// TwinCAT 3 PLC project segmentationDL
// ProgramVersion: 3.1.4026.10
// libraries:
//   Tc2_Standard, * (Beckhoff Automation GmbH)
//   Tc2_System, * (Beckhoff Automation GmbH)
//   Tc3_MlServer, * (Beckhoff Automation GmbH)
//   Tc3_Vision, * (Beckhoff Automation GmbH)
// project tree:
//   DUTs/ ST_modelInput.TcDUT, ST_modelOutput.TcDUT
//   GVLs/ constants.TcGVL
//   / PlcTask.TcTTO
//   POUs/Functions/ binarizeSegmentationMatrixFunction.TcPOU, contourSegmentationFunction.TcPOU, convertToBwFunction.TcPOU, flattenSegmentationMatrixFunction.TcPOU, imageNormalizationFunction.TcPOU, imageTilingFunction.TcPOU, imageToMatrixFunction.TcPOU, matrixToMaskFunction.TcPOU, nnPredictFunction.TcPOU, readImageFunction.TcPOU, reassembleImageFunction.TcPOU
//   POUs/Functions/Other/ binarizeSegmentationImageFunction.TcPOU, extractSingleTileFunction.TcPOU, flattenedTileToImageFunction.TcPOU, flattenMatrixFunction.TcPOU, flattenTileFunction.TcPOU, matrixToImageFunction.TcPOU
//   POUs/ MAIN.TcPOU
// real-time tasks:
//   TASK PlcTask: cycle T#10ms, priority 20, ADS port 350

CONFIGURATION segmentationDL
    RESOURCE PLC ON TwinCAT3
        TASK PlcTask(INTERVAL := T#10ms, PRIORITY := 20);
        PROGRAM MAIN WITH PlcTask : MAIN;
    END_RESOURCE
END_CONFIGURATION

// ---- DUTs/ST_modelInput.TcDUT
TYPE ST_modelInput :
STRUCT

	{attribute 'hide'} _header_DO_NOT_CHANGE : ARRAY[0..63] OF SINT := [-1,-112,120,86,52,18,-1,-1,1,-1,0,0,-1,-1,-112,-112,5,-37,-120,51,81,-94,-125,-64,-81,-119,-103,-51,-65,-118,48,-32,-5,44,-121,-88,-37,0,73,-109,92,-4,-120,92,99,42,-107,-53,64,-52,3,0,0,0,0,0,0,0,0,0,0,0,0,0];
	in_args_0 : ARRAY[0..0,0..287,0..215,0..0] OF REAL;

END_STRUCT
END_TYPE

// ---- DUTs/ST_modelOutput.TcDUT
TYPE ST_modelOutput :
STRUCT

	{attribute 'hide'} _header_DO_NOT_CHANGE : ARRAY[0..63] OF SINT := [-1,-112,120,86,52,18,-1,-1,1,-1,0,0,-1,-1,-112,-112,5,-37,-120,51,81,-94,-125,-64,-81,-119,-103,-51,-65,-118,48,-32,-5,44,-121,-88,-37,0,73,-109,92,-4,-120,92,99,42,-107,-53,64,-52,3,0,0,0,0,0,0,0,0,0,0,0,0,0];
	out_conv2d_14 : ARRAY[0..0,0..287,0..215,0..0] OF REAL;

END_STRUCT
END_TYPE

// ---- GVLs/constants.TcGVL
{attribute 'qualified_only'}
VAR_GLOBAL CONSTANT
	
	// Dimensions of the image
	IMG_WIDTH: UDINT := 1080;
	IMG_HEIGHT: UDINT := 1440;
	
	// Dimensions of the tile
	TILE_WIDTH: UDINT := 216;
	TILE_HEIGHT: UDINT := 288;
	
	// Total number of tiles
	NUM_TILES: UDINT := 25; 
	
END_VAR

// ---- POUs/MAIN.TcPOU
PROGRAM MAIN
VAR
	
	filePath: STRING := 'C:\Users\UserName\Desktop\visionFiles\images\000188.jpg'; // Change accordingly
	
	modelFilePath: STRING := 'C:\Users\UserName\Desktop\visionFiles\model\model.json'; // Change accordingly
	
	// Processing chain
	readImage: readImageFunction;
	convertToBw: convertToBwFunction;
	imageToMatrix: imageToMatrixFunction;
	imageNormalization: imageNormalizationFunction;
	imageTiling: imageTilingFunction;
	nnPredict: nnPredictFunction;
	reassembleImage: reassembleImageFunction;
	matrixToMask: matrixToMaskFunction;
	binarizeSegmentationMatrix: binarizeSegmentationMatrixFunction;
	contourSegmentation: contourSegmentationFunction;
	
	image: ITcVnImage;
	imageDisp: ITcVnDisplayableImage;
	
	segmentation: ITcVnImage;
	segmentationDisp: ITcVnDisplayableImage;
	
	contours: ITcVnImage;
	contoursDisp: ITcVnDisplayableImage;

	
	imageMatrix: ARRAY[1..constants.IMG_WIDTH, 1..constants.IMG_HEIGHT] OF REAL;
	tiles: ARRAY[1..constants.NUM_TILES, 1..constants.TILE_WIDTH, 1..constants.TILE_HEIGHT] OF REAL;
	
	segmentationTiles: ARRAY[1..constants.NUM_TILES, 1..constants.TILE_WIDTH, 1..constants.TILE_HEIGHT] OF REAL;
	segmentationMatrix: ARRAY[1..constants.IMG_WIDTH, 1..constants.IMG_HEIGHT] OF REAL;
	segmentationMatixBinarized: ARRAY[1..constants.IMG_WIDTH, 1..constants.IMG_HEIGHT] OF USINT;
	
	error: BOOL;
	hResult: HRESULT;

END_VAR

// Read the image
readImage(filePath := filePath,
		  image := image,
		  imageDisp := imageDisp,
		  error => error);
		  
// Convert the image to Black and White
convertToBw(image := image,
			imageDisp := imageDisp,
			start := readImage.finished,
			error => error);

// Extract the image values in the form of a matrix
imageToMatrix(image := image,
			  start := convertToBw.finished,
			  imageMatrix := imageMatrix,
			  error => error);

// Normalize image values from 0->255 to 0->1		  
imageNormalization(imageMatrix := imageMatrix,
					start := imageToMatrix.finished,
					error => error);
					
// Tile the image			  
imageTiling(tiles := tiles,
			imageMatrix := imageMatrix,
			start := imageNormalization.finished);
					
// Neural Network prediction
nnPredict(tiles := tiles,
		  modelFilePath := modelFilePath,
		  start := imageTiling.finished,
		  segmentationTiles => segmentationTiles);

// Reassembling tiles into an image matrix
reassembleImage(tiles := segmentationTiles,
				start := nnPredict.finished,
				imageMatrix => segmentationMatrix);
				
// Binarize the output of the neural network
binarizeSegmentationMatrix(segmentationMatrix := segmentationMatrix,
						   segmentationMatrixBinarized := segmentationMatixBinarized,
						   start := reassembleImage.finished);

// Use this to convert the segmentation matrix into a usable twincat image
matrixToMask(matrix := segmentationMatixBinarized,
			 image := segmentation,
			 imageDisp := segmentationDisp,
			 start := 	binarizeSegmentationMatrix.finished,
			 error => error);

// Plot the contour overlaid 
contourSegmentation(image := image,
					segmentationImage := segmentation,
					contoursImage := contours,
					contoursImageDisp := contoursDisp,
					minimumArea := 100,
					start := matrixToMask.finished,);

END_PROGRAM

// ---- POUs/Functions/readImageFunction.TcPOU
FUNCTION_BLOCK readImageFunction

VAR_IN_OUT
	image: ITcVnImage;
	imageDisp: ITcVnDisplayableImage;
END_VAR

VAR_INPUT
	filePath: STRING;
END_VAR

VAR_OUTPUT
	error: BOOL;
	finished: BOOL;
END_VAR


VAR
	readImageTrg: F_TRIG;	

	readImage: FB_VN_ReadImage;
	readImageCmd: BOOL := TRUE;
	
	imageRef: REFERENCE TO ITcVnImage;
	imageDispRef: REFERENCE TO ITcVnDisplayableImage;
	
	hResult: HRESULT;
	isImageRead: BOOL;
END_VAR

// Assign references
imageRef REF= image;
imageDispRef REF= imageDisp;

// Read the image
readImage(sFilePath := filePath,
          ipDestimage := imageRef,
          bRead := readImageCmd);
		 
// Trigger on when the image is read
readImageTrg(CLK := readImage.bBusy);

// If there is an error, latch onto it
IF readImage.bError THEN
    error := TRUE;
END_IF

// Reset the command after execution if needed for edge triggering
IF readImage.bBusy THEN
    readImageCmd := FALSE;
END_IF

// Raise a flag when the image has been read
IF (readImageTrg.Q) AND (NOT error) THEN
	isImageRead := TRUE;
END_IF

// Convert to a displayable image to view in the ADS Image View, if possible
IF (NOT error) AND (isImageRead) AND (NOT finished) THEN
	
    // Copy the image into a displayable one so that we can access it via the ADS Image Watch
    hResult := F_VN_CopyIntoDisplayableImage(ipSrcImage := image,
                                             ipDestImage := imageDispRef,
                                             hrPrev := hResult);

	// If there is an error, latch onto it
    IF FAILED(hResult) THEN
        error := TRUE;
    END_IF
	
	IF SUCCEEDED(hResult) THEN
		finished := TRUE;
	END_IF
	
END_IF

END_FUNCTION_BLOCK

// ---- POUs/Functions/convertToBwFunction.TcPOU
FUNCTION_BLOCK convertToBwFunction

VAR_IN_OUT
	image: ITcVnImage;
	imageDisp: ITcVnDisplayableImage;
END_VAR

VAR_INPUT
	start: BOOL;
END_VAR

VAR_OUTPUT
	error: BOOL;
	finished: BOOL := FALSE;
END_VAR


VAR

	originalImage: ITcVnImage;

	imageRef: REFERENCE TO ITcVnImage;
	imageDispRef: REFERENCE TO ITcVnDisplayableImage;
	
	hResult: HRESULT;
END_VAR

// Assign references
imageRef REF= image;
imageDispRef REF= imageDisp;
	
IF (start) AND (NOT error) AND (NOT finished) THEN
	
	originalImage := image;

	// Convert to black and white
	hResult := F_VN_ConvertColorSpace(ipSrcImage := image,
										ipDestImage := imageRef,
										eTransform := ETcVnColorSpaceTransform.TCVN_CST_RGB_TO_GRAY,
										hrPrev := hResult);
										
	// If there is an error, latch onto it
    IF FAILED(hResult) THEN
        error := TRUE;
    END_IF
	
	IF SUCCEEDED(hResult) THEN
		
		 // Copy the image into a displayable one so that we can access it via the ADS Image Watch
		hResult := F_VN_CopyIntoDisplayableImage(ipSrcImage := image,
											    	ipDestImage := imageDispRef,
											    	hrPrev := hResult);
	
		// If there is an error, latch onto it
		IF FAILED(hResult) THEN
			error := TRUE;
		END_IF
		
		IF SUCCEEDED(hResult) THEN
			finished := TRUE;
		END_IF
		
	END_IF
	
END_IF

END_FUNCTION_BLOCK

// ---- POUs/Functions/imageToMatrixFunction.TcPOU
FUNCTION_BLOCK imageToMatrixFunction

// See: https://infosys.beckhoff.com/english.php?content=../content/1033/tf7xxx_tc3_vision/6997345803.html&id=

VAR_IN_OUT
	imageMatrix: ARRAY[1..constants.IMG_WIDTH, 1..constants.IMG_HEIGHT] OF REAL;
END_VAR

VAR_INPUT
	image: ITcVnImage;
	start: BOOL;
END_VAR

VAR_OUTPUT
	error: BOOL;
	finished: BOOL := FALSE;
END_VAR

VAR
	
    nHeight     :   UDINT;
    nWidth      :   UDINT;
    y           :   UDINT;
    x           :   UDINT;
	
    pRow        :   POINTER TO USINT;
    nPixelValue :   USINT;
	
	hResult: HRESULT;
	
END_VAR

	
IF start AND (NOT finished) THEN
	
	// Retrieve the image width and height
	//hResult := F_VN_GetImageWidth(image, nWidth, hResult);
	//hResult := F_VN_GetImageHeight(image, nHeight, hResult);
	
	// Iterate every pixel of the image
	
	
	FOR y := 0 TO constants.IMG_HEIGHT - 1 DO
	
		// Get the pointer to the image row
		HRESULT := image.GetRowPointer(y, ADR(pRow));
		
		FOR x := 0 TO constants.IMG_WIDTH - 1 DO
			
			// Access the single pixel value
			nPixelValue := pRow[x]; 
			
			// Assign the pixel value to the image matrix
			imageMatrix[x+1, y+1] := nPixelValue; 
			
		END_FOR
	
		// It’s important to release the pointer. Otherwise there will be memory leaks.
		HRESULT := image.ReleaseRowPointer(ADR(pRow)); 
		
	END_FOR

	finished := TRUE;

END_IF

END_FUNCTION_BLOCK

// ---- POUs/Functions/imageNormalizationFunction.TcPOU
FUNCTION_BLOCK imageNormalizationFunction

VAR_IN_OUT
	imageMatrix: ARRAY[1..constants.IMG_WIDTH, 1..constants.IMG_HEIGHT] OF REAL;
END_VAR

VAR_INPUT
	start: BOOL;
END_VAR

VAR_OUTPUT
	error: BOOL;
	finished: BOOL := FALSE;
END_VAR

VAR
	x: UDINT;
	y: UDINT;
	normalizationFactor: REAL := 255.0;
END_VAR

	
IF (start) AND (NOT finished) THEN
	
	FOR x := 1 TO constants.IMG_WIDTH DO
		FOR y := 1 TO constants.IMG_HEIGHT DO
			
			imageMatrix[x, y] := imageMatrix[x, y] / normalizationfactor;
			
		END_FOR
	END_FOR
	
	finished := TRUE;
	 
END_IF

END_FUNCTION_BLOCK

// ---- POUs/Functions/imageTilingFunction.TcPOU
FUNCTION_BLOCK imageTilingFunction

VAR_IN_OUT
	tiles: ARRAY[1..constants.NUM_TILES, 1..constants.TILE_WIDTH, 1..constants.TILE_HEIGHT] OF REAL;
	start: BOOL;
END_VAR

VAR_INPUT
    imageMatrix: ARRAY[1..constants.IMG_WIDTH, 1..constants.IMG_HEIGHT] OF REAL;
END_VAR

VAR_OUTPUT
	finished: BOOL;
END_VAR

VAR
    tileRow: UDINT; // Row of the tile grid
    tileCol: UDINT; // Column of the tile grid
    currentTile: UDINT; // Counter for the tiles
    
    startX: UDINT; // X coordinate for the start of the tile
    startY: UDINT; // Y coordinate for the start of the tile
    X: UDINT; // X position within the tile
    Y: UDINT; // Y position within the tile
	
	nTilesHorizontal: UDINT;
	nTilesVertical: UDINT;
	
	
    
END_VAR


IF start AND NOT finished THEN
	
	// We start from the first tile
	currentTile := 1;
	
	// Finding how many tiles in the horizontal and vertical direction
	nTilesVertical := constants.IMG_HEIGHT / constants.TILE_HEIGHT;
	nTilesHorizontal := constants.IMG_WIDTH / constants.TILE_WIDTH;
	
	
	// Cycling on the tiles
	
	// Y
	FOR tileRow := 1 TO nTilesVertical DO
		
		// X
		FOR tileCol := 1 TO nTilesHorizontal DO
	
			// Determining the top left point coordinate of each tile
			startY := (tileRow - 1) * constants.TILE_HEIGHT + 1;
			startX := (tileCol - 1) * constants.TILE_WIDTH + 1;
			
			// Cycling on the pixels of the tile
			FOR X := 1 TO constants.TILE_WIDTH DO
				FOR Y := 1 TO constants.TILE_HEIGHT DO
					tiles[currentTile, X, Y] := imageMatrix[startX + X - 1, startY + Y - 1]; // Subtract 1 since the inner for loops add 1
				END_FOR
			END_FOR
	
			// Update the current tile
			currentTile := currentTile + 1;
	
		END_FOR
	END_FOR

	finished := TRUE;

END_IF

END_FUNCTION_BLOCK

// ---- POUs/Functions/nnPredictFunction.TcPOU
FUNCTION_BLOCK nnPredictFunction

// see: https://infosys.beckhoff.com/english.php?content=../content/1033/tf3820_tc3_machine_learning_server/17276127115.html&id=9003034378846799115

VAR_INPUT
	tiles: ARRAY[1..constants.NUM_TILES, 1..constants.TILE_WIDTH, 1..constants.TILE_HEIGHT] OF REAL;
	modelFilePath: STRING;
	start: BOOL;
END_VAR

VAR_OUTPUT
	segmentationTiles: ARRAY[1..constants.NUM_TILES, 1..constants.TILE_WIDTH, 1..constants.TILE_HEIGHT] OF REAL;
	finished: BOOL;
	error: BOOL;
END_VAR

VAR

	stModelInput: ST_modelInput;
	stModelOutput: ST_modelOutput;

	fbMlSvr: FB_MlSvrPrediction;
	
	n: UDINT := 1;
	x: UDINT;
	y: UDINT;
	
	nextTile: BOOL := TRUE;
	
END_VAR

// ===================================
// 1. Configuring the ML server
// ===================================

// Path to model  
fbMlSvr.stPredictionParameter.sMlModelFilePath := modelFilePath;

 // We want to execute the model on localsystem --> localhost                                     
fbMlSvr.stPredictionParameter.sMlSvrNetId := '127.0.0.1.1.1';

// Where to execute the model --> CPU
fbMlSVr.stPredictionParameter.eExecutionProvider := E_EXECUTIONPROVIDER.CPU; 

// Submit configuration request to the TcMlServer
fbMlSvr.Configure(nTimeout := 1000, nPriority:=0);

IF (fbMlSvr.bError) THEN
	error := TRUE;
END_IF


// ===================================================
// 2. Use the model for predictions
// ===================================================

// If the server is configured
IF (fbMlSvr.bConfigured) AND (start) AND (NOT finished) THEN
	
	// Cycling on the tiles, use an IF statement since it can take multiple PLC cycles
	IF n <= constants.NUM_TILES THEN
		
		// If it is time to process the next tile
		IF nextTile THEN
			
			nextTile := FALSE;
			
			// Format the tile for the model input
			FOR y := 1 TO constants.TILE_HEIGHT DO
				FOR x := 1 TO constants.TILE_WIDTH DO
					stModelInput.in_args_0[0, y-1, x-1, 0] := tiles[n, x, y];
				END_FOR
			END_FOR
			
		END_IF
		
		// Predict
		IF fbMlSvr.Predict(pDataIn := ADR(stModelInput), 
						   nDataInSize := SIZEOF(stModelInput), 
						   pDataOut := ADR(stModelOutput), 
						   nDataOutSize := SIZEOF(stModelOutput),
						   nTimeout := 10000,
						   nPriority := 0) THEN
						   
			// Reassemble output
			FOR y := 1 TO constants.TILE_HEIGHT DO
				FOR x := 1 TO constants.TILE_WIDTH DO
					segmentationTiles[n, x, y] := stModelOutput.out_conv2d_14[0, y-1, x-1, 0];
				END_FOR
			END_FOR
					
			// Go to next tile	   
			nextTile := TRUE;
			n := n+1;
							
		END_IF
		
	END_IF
	
END_IF	

// When it has finished processing all the tiles, raise a flag
finished := (n = constants.NUM_TILES+1);

END_FUNCTION_BLOCK

// ---- POUs/Functions/reassembleImageFunction.TcPOU
FUNCTION_BLOCK reassembleImageFunction

VAR_IN_OUT
    tiles: ARRAY[1..constants.NUM_TILES, 1..constants.TILE_WIDTH, 1..constants.TILE_HEIGHT] OF REAL;
    start: BOOL;
END_VAR

VAR_OUTPUT
    imageMatrix: ARRAY[1..constants.IMG_WIDTH, 1..constants.IMG_HEIGHT] OF REAL;
    finished: BOOL;
END_VAR

VAR
    tileRow: UDINT;
    tileCol: UDINT;
    currentTile: UDINT;

    startX: UDINT;
    startY: UDINT;
    X: UDINT;
    Y: UDINT;

    nTilesHorizontal: UDINT;
    nTilesVertical: UDINT;
	
END_VAR


IF start AND NOT finished THEN
	
	// We start from the first tile
	currentTile := 1;
	
	// Finding how many tiles in the horizontal and vertical direction
	nTilesVertical := constants.IMG_HEIGHT / constants.TILE_HEIGHT;
	nTilesHorizontal := constants.IMG_WIDTH / constants.TILE_WIDTH;
	
	
	// Cycling on the tiles
	
	// Y
	FOR tileRow := 1 TO nTilesVertical DO
		
		// X
		FOR tileCol := 1 TO nTilesHorizontal DO
	
			// Determining the top left point coordinate of each tile
			startY := (tileRow - 1) * constants.TILE_HEIGHT + 1;
			startX := (tileCol - 1) * constants.TILE_WIDTH + 1;
			
			// Cycling on the pixels of the tile
			FOR X := 1 TO constants.TILE_WIDTH DO
				FOR Y := 1 TO constants.TILE_HEIGHT DO
					imageMatrix[startX + X - 1, startY + Y - 1] := tiles[currentTile, X, Y]; // Subtract 1 since the inner for loops add 1
				END_FOR
			END_FOR
	
			// Update the current tile
			currentTile := currentTile + 1;
	
		END_FOR
	END_FOR

	finished := TRUE;

END_IF

END_FUNCTION_BLOCK

// ---- POUs/Functions/matrixToMaskFunction.TcPOU
FUNCTION_BLOCK matrixToMaskFunction

VAR_IN_OUT
	matrix: ARRAY[1..constants.IMG_WIDTH, 1..constants.IMG_HEIGHT] OF USINT;
	image: ITcVnImage;
	imageDisp: ITcVnDisplayableImage;
END_VAR

VAR_INPUT
	start: BOOL;
END_VAR

VAR_OUTPUT
	error: BOOL;
	finished: BOOL;
END_VAR

VAR
	flattenSegmentationMatrix: flattenSegmentationMatrixFunction;
	hResult: HRESULT;
	ePixelType: ETcVnElementType;
	imageDispRef: REFERENCE TO ITcVnDisplayableImage;
	flattenedMatrix: ARRAY[1..constants.IMG_WIDTH*constants.IMG_HEIGHT] OF USINT;
	flattenedMatrixPtr: POINTER TO ARRAY[1..constants.IMG_WIDTH*constants.IMG_HEIGHT] OF USINT;
END_VAR

IF (start) AND (NOT finished) THEN
	
	imageDispRef REF= imageDisp;
	
	// Flatten the matrix
	flattenSegmentationMatrix(matrix := matrix,
							  start := start,
							  flattenedMatrix := flattenedMatrix);
				  
	// When it finished flattening, we create the image object of Twincat Vision
	IF flattenSegmentationMatrix.finished THEN
		
		flattenedMatrixPtr := ADR(flattenedMatrix);
		

		F_VN_CreateImageFromArray(nWidth := constants.IMG_WIDTH,
								  nHeight := constants.IMG_HEIGHT,
								  nChannelNum := 1, 					// Black and white
								  ipImage := image,
								  pData := flattenedMatrixPtr,
								  ePixelType := ETcVnElementType.TCVN_ET_USINT,
								  hrPrev := hResult);
								  
		IF FAILED(hResult) THEN
			error := TRUE;
		END_IF
								  
		IF SUCCEEDED(hResult) THEN
				  
			// Copy the image into a displayable one so that we can access it via the ADS Image Watch
			hResult := F_VN_CopyIntoDisplayableImage(ipSrcImage := image,
													 ipDestImage := imageDispRef,
													 hrPrev := hResult);
			IF FAILED(hResult) THEN
				error := TRUE;
			END_IF
			IF SUCCEEDED(hResult) THEN 
				finished := TRUE;
			END_IF
					
		END_IF
	
	END_IF
	
END_IF

END_FUNCTION_BLOCK

// ---- POUs/Functions/flattenSegmentationMatrixFunction.TcPOU
FUNCTION_BLOCK flattenSegmentationMatrixFunction
VAR_INPUT
	matrix: ARRAY[1..constants.IMG_WIDTH, 1..constants.IMG_HEIGHT] OF USINT;
	start: BOOL;
END_VAR

VAR_IN_OUT
	flattenedMatrix: ARRAY[1..constants.IMG_WIDTH*constants.IMG_HEIGHT] OF USINT;
END_VAR

VAR_OUTPUT
	finished: BOOL;
END_VAR


VAR
	i: UDINT;
	x: UDINT;
	y: UDINT;
END_VAR


IF (start) AND (NOT finished) THEN
	
	// We start from one
	i := 1;
	
	// First we have to cycle on the y,
	// as the flattened vector is expected to be set up in this way
	FOR y := 1 TO constants.IMG_HEIGHT DO
		
		// Then we have to cycle on the x
		FOR x := 1 TO constants.IMG_WIDTH DO
			flattenedMatrix[i] := matrix[x, y];
			i := i+1;
		END_FOR
	END_FOR

	finished := TRUE;

END_IF

END_FUNCTION_BLOCK

// ---- POUs/Functions/binarizeSegmentationMatrixFunction.TcPOU
FUNCTION_BLOCK binarizeSegmentationMatrixFunction

VAR_INPUT
	segmentationMatrix: ARRAY[1..constants.IMG_WIDTH, 1..constants.IMG_HEIGHT] OF REAL;
	start: BOOL;
END_VAR

VAR_OUTPUT
	finished: BOOL;
END_VAR

VAR_IN_OUT
	segmentationMatrixBinarized: ARRAY[1..constants.IMG_WIDTH, 1..constants.IMG_HEIGHT] OF USINT; // From 0 to 255
END_VAR

VAR
	x: UDINT;
	y: UDINT;
END_VAR

IF start AND (NOT finished) THEN

	FOR y := 1 TO constants.IMG_HEIGHT DO
		FOR x := 1 TO constants.IMG_WIDTH DO
			
			IF segmentationMatrix[x, y] > 0.5 THEN // 0.5 is the threhsold of the neural network
				segmentationMatrixBinarized[x, y] := 255;
			ELSE
				segmentationMatrixBinarized[x, y] := 0;
			END_IF
			
		END_FOR
	END_FOR
	
	finished := TRUE;
	
END_IF

END_FUNCTION_BLOCK

// ---- POUs/Functions/contourSegmentationFunction.TcPOU
FUNCTION_BLOCK contourSegmentationFunction

VAR_INPUT
	image: ITcVnImage; // The image "with the background"
	segmentationImage: ITcVnImage; // The twincat image which contains the binarized segmentation mask
	start: BOOL;
	minimumArea: LREAL; // Minimum area for a defect for filtering small imprecisions
END_VAR

VAR_IN_OUT
	contoursImage: ITcVnImage; // The image in which to display the segmentation
	contoursImageDisp: ITcVnDisplayableImage;
END_VAR


VAR_OUTPUT
	finished: BOOL;
END_VAR

VAR

	contoursImageRef: REFERENCE TO ITcVnImage;
	contoursImageDispRef: REFERENCE TO ITcVnDisplayableImage;
	imageRgb: ITcVnImage;
	imageRgbRef: REFERENCE TO ITcVnImage;

	ipContourListRef: REFERENCE TO ITcVnContainer;
	ipContour: ITcVnContainer;
	ipIterator: ITcVnForwardIterator; // To iterate within the container of the contours
	hResult: HRESULT;
	aColorRed: TcVnVector4_LREAL := [255,0,0];
	ipContourList: ITcVnContainer;
	
	fArea: LREAL; // The found area of from the contour
	aCenter: TcVnPoint2_LREAL; // The center of the contour

	oldCenter: TcVnPoint2_LREAL;
	distanceBetweenDefects: LREAL := 100;
	deltaX: LREAL;
	
END_VAR

ipContourListRef REF= ipContourList;
contoursImageRef REF= contoursImage;
contoursImageDispRef REF= contoursImageDisp;
imageRgbRef REF= imageRgb;

IF (start) AND (NOT finished) THEN
	
	// Pass from grayscale to RGB 
	hResult := F_VN_ConvertColorSpace(ipSrcImage := image,
									  ipDestImage := imageRgbRef,
									  eTransform := ETcVnColorSpaceTransform.TCVN_CST_GRAY_TO_RGB,
							     	  hrPrev := hResult);
		
	// Copy the original image into the one with the contours so to have the background
	hResult := F_VN_CopyImage(imageRgb, contoursImageRef, hResult);

	// Find the contours 
	hResult := F_VN_FindContours(ipSrcImage := segmentationImage,
								 ipContours := ipContourListRef,
					  			 hrPrev := hResult);

	// Convert the contours into a displayble image if (1) we succeeded and (2) if we have not reached the end of the container
	hResult := F_VN_GetForwardIterator(ipContourListRef, ipIterator, hResult);
	WHILE SUCCEEDED(hResult) AND_THEN ipIterator.CheckIfEnd() <> S_OK DO
		
		hResult := F_VN_GetContainer(ipIterator, ipContour, hResult);
		hResult := F_VN_IncrementIterator(ipIterator, hResult);
		hResult := F_VN_ContourArea(ipContour, fArea, hResult);
		
		// Plot only if it is bigger than the minimum area
		IF fArea >=minimumArea THEN
			
			// Plot the contour
			hResult := F_VN_DrawContours(ipContour, -1, contoursImage, aColorRed, 3, hResult);
			
			// Find the center of the contour
			hResult := F_VN_ContourCenterOfMass(ipContour, aCenter, hResult);
			
			// Put a new text only if the center of mass is far enough
			IF (ABS(aCenter[0]-oldCenter[0]) + ABS(aCenter[1]-oldCenter[1])) > distanceBetweenDefects THEN
				
				// Putting the label either left or right
				IF aCenter[0] > constants.IMG_WIDTH/2 THEN
					deltaX := +50;
				ELSE
					deltaX := -200;
				END_IF

				// Plot the text
				hResult := F_VN_PutText(sText := 'DEFECT', 
										ipDestImage := contoursImage,
										nX := LREAL_TO_UDINT(aCenter[0]+deltaX), 
										nY := LREAL_TO_UDINT(aCenter[1]),
										eFontType := ETcVnFontType.TCVN_FT_HERSHEY_TRIPLEX,
										fFontScale := 1,
										aColor := aColorRed,
										hrPrev := hResult);
				
			END_IF
			
			oldCenter := aCenter;
			

		END_IF

	END_WHILE
	
	// Copy the image into a displayable one so that we can access it via the ADS Image Watch
    hResult := F_VN_CopyIntoDisplayableImage(ipSrcImage := contoursImage,
                                             ipDestImage := contoursImageDispRef,
                                             hrPrev := hResult);
	
	IF SUCCEEDED(hResult) THEN
		finished := TRUE;
	END_IF
	
END_IF

END_FUNCTION_BLOCK

// ---- POUs/Functions/Other/binarizeSegmentationImageFunction.TcPOU
FUNCTION_BLOCK binarizeSegmentationImageFunction
VAR_IN_OUT
	segmentationImage: ITcVnImage;
    segmentationImageBinarized: ITcVnImage;
	segmentationImageBinarizedDisp: ITcVnDisplayableImage;
END_VAR

VAR_INPUT
	start: BOOL;
END_VAR

VAR_OUTPUT
	finished: BOOL;
END_VAR

VAR
	segmentationImageBinarizedRef: REFERENCE TO ITcVnImage;
	
	fThreshold: LREAL := 0.5;
    fMaxValue: LREAL := 255; // 255 is the maximum representable integer in the 8 bit color space
    eThresholdType: ETcVnThresholdType := ETcVnThresholdType.TCVN_TT_BINARY;
    hResult: HRESULT;
END_VAR

segmentationImageBinarizedRef REF= segmentationImageBinarized;

IF start AND (NOT finished) THEN
	
	hResult := F_VN_Threshold(ipSrcImage := segmentationImage,
							  ipDestImage := segmentationImageBinarizedRef,
							  fThreshold := fThreshold, 
							  fMaxValue := fMaxValue,
							  eThresholdType := eThresholdType,
							  hrPrev := hResult);
	
	IF SUCCEEDED(hResult) THEN
		
		 // Copy the image into a displayable one so that we can access it via the ADS Image Watch
		hResult := F_VN_CopyIntoDisplayableImage(ipSrcImage := segmentationImageBinarized,
											     ipDestImage := segmentationImageBinarizedDisp,
											     hrPrev := hResult);
												 
		IF SUCCEEDED(hResult) THEN
			finished := TRUE;
		END_IF
		
	END_IF
	
					  
END_IF

END_FUNCTION_BLOCK

// ---- POUs/Functions/Other/extractSingleTileFunction.TcPOU
FUNCTION_BLOCK extractSingleTileFunction

VAR_IN_OUT
	tile: ARRAY[1..constants.TILE_WIDTH, 1..constants.TILE_HEIGHT] OF REAL;
END_VAR

VAR_INPUT
	tiles: ARRAY[1..constants.NUM_TILES, 1..constants.TILE_WIDTH, 1..constants.TILE_HEIGHT] OF REAL; 
	tileToExtract: UDINT; // Assuming it is within the number of admissible tiles
	start: BOOL;
END_VAR

VAR_OUTPUT
	finished: BOOL;
END_VAR

VAR
	x: UDINT;
	y: UDINT;
END_VAR

IF start AND (NOT finished) THEN
	
	
	FOR x := 1 TO constants.TILE_WIDTH DO
		FOR y := 1 TO constants.TILE_HEIGHT DO
			
			tile[x, y] := tiles[tileToExtract, x, y];
			
		END_FOR;
	END_FOR
	
	finished := TRUE;
	
END_IF

END_FUNCTION_BLOCK

// ---- POUs/Functions/Other/flattenedTileToImageFunction.TcPOU
FUNCTION_BLOCK flattenedTileToImageFunction

VAR_IN_OUT
	image: ITcVnImage;
	imageDisp: ITcVnDisplayableImage;
	flattenedTile: ARRAY[1..constants.TILE_WIDTH*constants.TILE_HEIGHT] OF REAL;
END_VAR

VAR_INPUT
	start: BOOL;
END_VAR

VAR
	finished: BOOL;
	hResult: HRESULT;
	imageDispRef: REFERENCE TO ITcVnDisplayableImage;
	flattenedTilePtr: POINTER TO ARRAY[1..constants.TILE_WIDTH*constants.TILE_HEIGHT] OF REAL;
END_VAR

IF (start) AND (NOT finished) THEN
	
	imageDispRef REF= imageDisp;
	
	flattenedTilePtr := ADR(flattenedTile);
	
	F_VN_CreateImageFromArray(nWidth := constants.TILE_WIDTH,
							  nHeight := constants.TILE_HEIGHT,
							  nChannelNum := 1, 					// Black and white
							  ipImage := image,
							  pData := flattenedTilePtr,
							  ePixelType := ETcVnElementType.TCVN_ET_REAL,
							  hrPrev := hResult);
							  
	IF SUCCEEDED(hResult) THEN
			  
		// Copy the image into a displayable one so that we can access it via the ADS Image Watch
		hResult := F_VN_CopyIntoDisplayableImage(ipSrcImage := image,
												 ipDestImage := imageDispRef,
												 hrPrev := hResult);
		IF SUCCEEDED(hResult) THEN 
			finished := TRUE;
		END_IF
		
		
	END_IF
	
END_IF

END_FUNCTION_BLOCK

// ---- POUs/Functions/Other/flattenMatrixFunction.TcPOU
FUNCTION_BLOCK flattenMatrixFunction
VAR_INPUT
	matrix: ARRAY[1..constants.IMG_WIDTH, 1..constants.IMG_HEIGHT] OF REAL;
	start: BOOL;
END_VAR

VAR_IN_OUT
	flattenedMatrix: ARRAY[1..constants.IMG_WIDTH*constants.IMG_HEIGHT] OF REAL;
END_VAR

VAR_OUTPUT
	finished: BOOL;
END_VAR


VAR
	i: UDINT;
	x: UDINT;
	y: UDINT;
END_VAR


IF (start) AND (NOT finished) THEN
	
	// We start from one
	i := 1;
	
	// First we have to cycle on the y,
	// as the flattened vector is expected to be set up in this way
	FOR y := 1 TO constants.IMG_HEIGHT DO
		
		// Then we have to cycle on the x
		FOR x := 1 TO constants.IMG_WIDTH DO
			flattenedMatrix[i] := matrix[x, y];
			i := i+1;
		END_FOR
	END_FOR

	finished := TRUE;

END_IF

END_FUNCTION_BLOCK

// ---- POUs/Functions/Other/flattenTileFunction.TcPOU
FUNCTION_BLOCK flattenTileFunction
VAR_INPUT
	tile: ARRAY[1..constants.TILE_WIDTH, 1..constants.TILE_HEIGHT] OF REAL;
	start: BOOL;
END_VAR

VAR_IN_OUT
	flattenedTile: ARRAY[1..constants.TILE_WIDTH*constants.TILE_HEIGHT] OF REAL;
END_VAR

VAR_OUTPUT
	finished: BOOL;
END_VAR

VAR
	i: UDINT;
	x: UDINT;
	y: UDINT;
END_VAR


IF (start) AND (NOT finished) THEN
	
	// We start from one
	i := 1;
		
	// First we have to cycle on the y
	FOR y := 1 TO constants.TILE_HEIGHT DO
		// Then we have to cycle no the x --> the flattened array is expected in this form
		FOR x := 1 TO constants.TILE_WIDTH DO
			flattenedTile[i] := tile[x, y];
			i := i+1;
		END_FOR
	END_FOR

	finished := TRUE;

END_IF

END_FUNCTION_BLOCK

// ---- POUs/Functions/Other/matrixToImageFunction.TcPOU
FUNCTION_BLOCK matrixToImageFunction

VAR_IN_OUT
	matrix: ARRAY[1..constants.IMG_WIDTH, 1..constants.IMG_HEIGHT] OF REAL;
	image: ITcVnImage;
	imageDisp: ITcVnDisplayableImage;
END_VAR

VAR_INPUT
	start: BOOL;
END_VAR

VAR_OUTPUT
	error: BOOL;
	finished: BOOL;
END_VAR

VAR
	flattenMatrix: flattenMatrixFunction;
	hResult: HRESULT;
	ePixelType: ETcVnElementType;
	imageDispRef: REFERENCE TO ITcVnDisplayableImage;
	flattenedMatrix: ARRAY[1..constants.IMG_WIDTH*constants.IMG_HEIGHT] OF REAL;
	flattenedMatrixPtr: POINTER TO ARRAY[1..constants.IMG_WIDTH*constants.IMG_HEIGHT] OF REAL;
END_VAR

IF (start) AND (NOT finished) THEN
	
	imageDispRef REF= imageDisp;
	
	// Flatten the matrix
	flattenMatrix(matrix := matrix,
				  start := start,
				  flattenedMatrix := flattenedMatrix);
				  
	// When it finished flattening, we create the image object of Twincat Vision
	IF flattenMatrix.finished THEN
		
		flattenedMatrixPtr := ADR(flattenedMatrix);
		

		F_VN_CreateImageFromArray(nWidth := constants.IMG_WIDTH,
								  nHeight := constants.IMG_HEIGHT,
								  nChannelNum := 1, 					// Black and white
								  ipImage := image,
								  pData := flattenedMatrixPtr,
								  ePixelType := ETcVnElementType.TCVN_ET_REAL,
								  hrPrev := hResult);
								  
		IF FAILED(hResult) THEN
			error := TRUE;
		END_IF
								  
		IF SUCCEEDED(hResult) THEN
				  
			// Copy the image into a displayable one so that we can access it via the ADS Image Watch
			hResult := F_VN_CopyIntoDisplayableImage(ipSrcImage := image,
													 ipDestImage := imageDispRef,
													 hrPrev := hResult);
			IF FAILED(hResult) THEN
				error := TRUE;
			END_IF
			IF SUCCEEDED(hResult) THEN 
				finished := TRUE;
			END_IF
					
		END_IF
	
	END_IF
	
END_IF

END_FUNCTION_BLOCK
